FUNCTION_BLOCK xPlanarErrorHandling
VAR_INPUT
END_VAR
VAR_OUTPUT
END_VAR
VAR
	Running			: BYTE;
	
	i				: BYTE;
	State			: BYTE;
	CommandDone		: BOOL;
	
	ResetDone		: BOOL;
	ErrorDetected	: BOOL;
	ErrorCount		: INT;
	ErrorTrigger	: R_Trig;
END_VAR


Running := Running + 1;

DetectErrors();

ErrorCounter();

ResetErrors();

METHOD DetectErrors : BOOL
VAR_INPUT
END_VAR

FOR i := 1 TO xPlanarLink.MoverCount DO
	IF xPlanarLink.PlanarMover[i].Error THEN
		ErrorDetected := TRUE;
	END_IF
END_FOR
END_METHOD

METHOD ErrorCounter : BOOL
VAR_INPUT
END_VAR

ErrorTrigger(CLK := ErrorDetected);

IF ErrorTrigger.Q THEN
	ErrorCount := ErrorCount + 1;
END_IF
END_METHOD

METHOD ResetErrors : BOOL
VAR_INPUT
END_VAR

IF ErrorDetected THEN

	CASE State OF
		
		0: 
			ResetDone := FALSE;
			FOR i := 1 TO xPlanarLink.MoverCount DO
				xPlanarLink.PlanarMover[i].Reset(xPlanarLink.PlanarFeedback[i]);
			END_FOR
			State := 1;
		
		1:	
			IF xPlanarLink.PlanarFeedback[1].Done AND xPlanarLink.PlanarFeedback[2].Done THEN
				CommandDone := FALSE;
				State := 2;
			END_IF
				
		2:
			ResetDone := TRUE;
		
	END_CASE	


END_IF
END_METHOD

END_FUNCTION_BLOCK

(* stored: Version 1.1.0.1, ProductVersion 3.1.4024.12
   POU xPlanarErrorHandling: Id {55eda779-33a1-444a-9c3a-a8daf9dafe63}, SpecialFunc None
   Method DetectErrors: Id {010aa0d9-eca0-4038-9ff3-7c9c3593edec}
   Method ErrorCounter: Id {7ad35de8-3e39-49fa-9986-7e86c77060b7}
   Method ResetErrors: Id {8372b3d2-7b21-40df-b1c7-03c57c4fc61a} *)
